// TIA Portal V19 export
FUNCTION "ReadRecord" : Void   // FC17, LAD
TITLE = Acrhive Read Record
// stored: SetENOAutomatically false
   VAR_INPUT
      ArchiveType : USInt;
      Exe : Bool;
      RecordToRead : Int;
   END_VAR
   VAR_OUTPUT
      Record : Variant;
      Done : Bool;
      Error : Bool;
   END_VAR
   VAR_TEMP
      ReadResult : Int;
      ReadInProgress : Bool;
   END_VAR
BEGIN

REGION Network 1 (SCL): Read Record
   CASE #ArchiveType OF
       0:  #ReadResult := READ_DBL(REQ := #Exe, SRCBLK := "PPrfArchive1".PRG[#RecordToRead], BUSY => #ReadInProgress, DSTBLK => #Record);
       1:  CASE #RecordToRead OF
               1..100:
                   #ReadResult := READ_DBL(REQ := #Exe, SRCBLK := "G.PPrgArchive1".PRG[#RecordToRead], BUSY => #ReadInProgress, DSTBLK => #Record);
               101..200:
                   #ReadResult := READ_DBL(REQ := #Exe, SRCBLK := "G.PPrgArchive2".PRG[#RecordToRead], BUSY => #ReadInProgress, DSTBLK => #Record);
               201..300:
                   #ReadResult := READ_DBL(REQ := #Exe, SRCBLK := "G.PPrgArchive3".PRG[#RecordToRead], BUSY => #ReadInProgress, DSTBLK => #Record);
               301..400:
                   #ReadResult := READ_DBL(REQ := #Exe, SRCBLK := "G.PPrgArchive4".PRG[#RecordToRead], BUSY => #ReadInProgress, DSTBLK => #Record);
               401..500:
                   #ReadResult := READ_DBL(REQ := #Exe, SRCBLK := "G.PPrgArchive5".PRG[#RecordToRead], BUSY => #ReadInProgress, DSTBLK => #Record);
               501..600:
                   #ReadResult := READ_DBL(REQ := #Exe, SRCBLK := "G.PPrgArchive6".PRG[#RecordToRead], BUSY => #ReadInProgress, DSTBLK => #Record);
               601..700:
                   #ReadResult := READ_DBL(REQ := #Exe, SRCBLK := "G.PPrgArchive7".PRG[#RecordToRead], BUSY => #ReadInProgress, DSTBLK => #Record);
               701..800:
                   #ReadResult := READ_DBL(REQ := #Exe, SRCBLK := "G.PPrgArchive8".PRG[#RecordToRead], BUSY => #ReadInProgress, DSTBLK => #Record);
               801..900:
                   #ReadResult := READ_DBL(REQ := #Exe, SRCBLK := "G.PPrgArchive9".PRG[#RecordToRead], BUSY => #ReadInProgress, DSTBLK => #Record);
               901..1000:
                   #ReadResult := READ_DBL(REQ := #Exe, SRCBLK := "G.PPrgArchive10".PRG[#RecordToRead], BUSY => #ReadInProgress, DSTBLK => #Record);
               1001..1100:
                   #ReadResult := READ_DBL(REQ := #Exe, SRCBLK := "G.PPrgArchive11".PRG[#RecordToRead], BUSY => #ReadInProgress, DSTBLK => #Record);
               1101..1200:
                   #ReadResult := READ_DBL(REQ := #Exe, SRCBLK := "G.PPrgArchive12".PRG[#RecordToRead], BUSY => #ReadInProgress, DSTBLK => #Record);
               1201..1300:
                   #ReadResult := READ_DBL(REQ := #Exe, SRCBLK := "G.PPrgArchive13".PRG[#RecordToRead], BUSY => #ReadInProgress, DSTBLK => #Record);
               1301..1400:
                   #ReadResult := READ_DBL(REQ := #Exe, SRCBLK := "G.PPrgArchive14".PRG[#RecordToRead], BUSY => #ReadInProgress, DSTBLK => #Record);
               1401..1500:
                   #ReadResult := READ_DBL(REQ := #Exe, SRCBLK := "G.PPrgArchive15".PRG[#RecordToRead], BUSY => #ReadInProgress, DSTBLK => #Record);
               1501..1600:
                   #ReadResult := READ_DBL(REQ := #Exe, SRCBLK := "G.PPrgArchive16".PRG[#RecordToRead], BUSY => #ReadInProgress, DSTBLK => #Record);
               1601..1700:
                   #ReadResult := READ_DBL(REQ := #Exe, SRCBLK := "G.PPrgArchive17".PRG[#RecordToRead], BUSY => #ReadInProgress, DSTBLK => #Record);
               1701..1800:
                   #ReadResult := READ_DBL(REQ := #Exe, SRCBLK := "G.PPrgArchive18".PRG[#RecordToRead], BUSY => #ReadInProgress, DSTBLK => #Record);
               1801..1900:
                   #ReadResult := READ_DBL(REQ := #Exe, SRCBLK := "G.PPrgArchive19".PRG[#RecordToRead], BUSY => #ReadInProgress, DSTBLK => #Record);
               1901..2000:
                   #ReadResult := READ_DBL(REQ := #Exe, SRCBLK := "G.PPrgArchive20".PRG[#RecordToRead], BUSY => #ReadInProgress, DSTBLK => #Record);
           END_CASE;
   END_CASE;
   #Done := #Exe AND #ReadResult = 0 AND NOT #ReadInProgress;
   #Error := #Exe AND #ReadResult <> 0 AND NOT #ReadInProgress;
END_REGION
END_FUNCTION
